TYPE u_SM6020_caudal :
UNION
	caudal: ARRAY[0..1] OF BYTE;
	icaudal			:INT;
END_UNION
END_TYPE

(* stored: Version 1.1.0.1, ProductVersion 3.1.4024.12
   DUT u_SM6020_caudal: Id {66af79c1-0813-4e58-8ffb-e7907026bf8c} *)
